PROGRAM P_Demo_FB_GetAdaptersInfo
VAR
    fbFB_GetAdaptersInfo : FB_GetAdaptersInfo; // FB_GetAdaptersInfo 实例
    sNetID               : T_AmsNetID := '';
    bExecute             : BOOL := FALSE;
    tTimeout             : TIME := DEFAULT_ADS_TIMEOUT;
    bBusy                : BOOL;
    bError               : BOOL;
    nErrID               : UDINT;
    arrAdapters          : ARRAY[0..MAX_LOCAL_ADAPTERS] OF ST_IpAdapterInfo;
    nCount               : UDINT;
    nGet                 : UDINT;
END_VAR

// =============================================================================
// 场景：FB_GetAdaptersInfo 的最小可编译演示——所有 VAR_INPUT 均以 doc/PDF 中真实引脚名调用。
//       业务侧请在线 monitor / 在线写值触发对应输入，看输出端 monitor 结果。
//
// 价值：保证示例 ST 代码所有引脚名与 FB_GetAdaptersInfo 的 VAR_INPUT/VAR_OUTPUT 一致，
//       Add Existing Item (.TcPOU) → 编译 → 登录 流程能跑通，作为 hand-curated 例程
//       的脚手架。
//
// 验证步骤：
//   1. 引用 Tc2_Utilities（及其依赖 Tc2_System）
//   2. 右键 PLC 项目下 POUs 文件夹 → Add → Existing Item → 选本 .TcPOU 文件 → OK → 编译、登录
//   3. 在线对 VAR_INPUT 写入合适触发值（典型 bExecute / RUN / START 上升沿）
//   4. 在线 monitor VAR_OUTPUT 观察 FB 反应
// =============================================================================

fbFB_GetAdaptersInfo(
    sNetID := sNetID,
    bExecute := bExecute,
    tTimeout := tTimeout,
    bBusy => bBusy,
    bError => bError,
    nErrID => nErrID,
    arrAdapters => arrAdapters,
    nCount => nCount,
    nGet => nGet
);

END_PROGRAM

(* stored: Version 1.1.0.1, ProductVersion 3.1.4024.5
   POU P_Demo_FB_GetAdaptersInfo: Id {4ceca5fa-4f31-57ae-a2ad-3fcabd182dc7}, SpecialFunc None *)
